// TIA Portal V16 program export: 1 tag tables, 0 data types, 0 data blocks, 1 code blocks (in call order from the OBs), 0 instance data blocks

VAR_GLOBAL   // PLC tag table "PuShButton_Interlocking"
   Stop AT %I0.0 : Bool;
   Forward_Start AT %I0.1 : Bool;
   Forward_Motor AT %Q0.0 : Bool;
   Back_Start AT %I0.2 : Bool;
   Back_Motor AT %Q0.1 : Bool;
END_VAR

ORGANIZATION_BLOCK "PushButton_Interlocking"   // OB1, LAD, ProgramCycle
TITLE = "Main Program Sweep (Cycle)"
{ S7_Optimized_Access := 'TRUE' }
VERSION : 0.1
// stored: AutoNumber true, IsIECCheckEnabled false, SetENOAutomatically false
   VAR_INPUT
      Initial_Call : Bool;   // Initial call of this OB
      Remanence : Bool;   // =True, if remanent data are available
   END_VAR
BEGIN

REGION Network 1
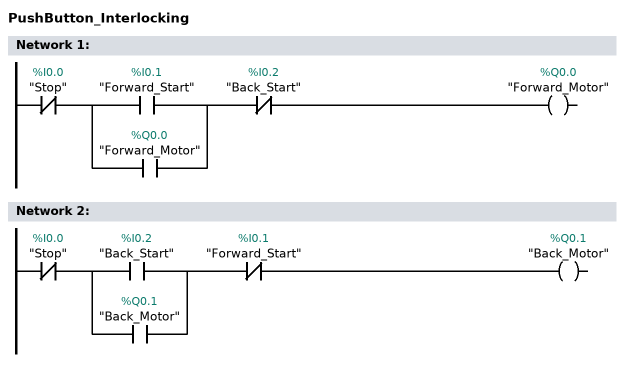
   RUNG wire#powerrail
      I_Contact( "Stop" )
      wire#w1
      Contact( "Forward_Start" )
      wire#w2
      I_Contact( "Back_Start" )
      Coil( "Forward_Motor" )
   END_RUNG
   RUNG wire#w1
      Contact( "Forward_Motor" )
   END_RUNG wire#w2
   // the same network as SCL:
   "Forward_Motor" := NOT "Stop" AND ("Forward_Start" OR "Forward_Motor") AND NOT "Back_Start";
END_REGION

REGION Network 2
   RUNG wire#powerrail
      I_Contact( "Stop" )
      wire#w1
      Contact( "Back_Start" )
      wire#w2
      I_Contact( "Forward_Start" )
      Coil( "Back_Motor" )
   END_RUNG
   RUNG wire#w1
      Contact( "Back_Motor" )
   END_RUNG wire#w2
   // the same network as SCL:
   "Back_Motor" := NOT "Stop" AND ("Back_Start" OR "Back_Motor") AND NOT "Forward_Start";
END_REGION
END_ORGANIZATION_BLOCK
